Omron CX-Programmer project NewProject (CX-Programmer 9.73)

# PLC NewPLC1: CP1E N30

## Program NewProgram1 (cyclic task 0)

### Section Section1

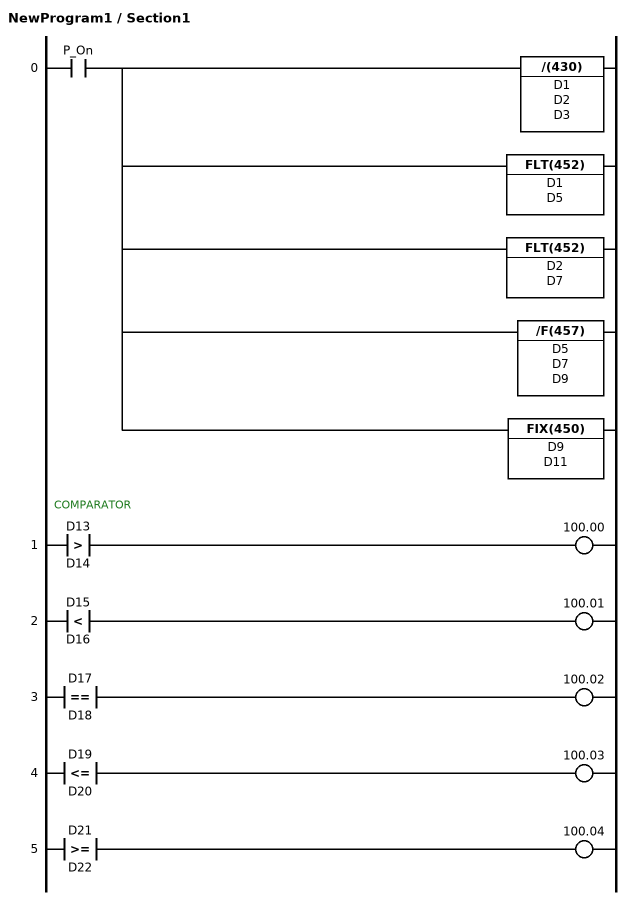
; rung 0
LD P_On
/(430) D1 D2 D3
FLT(452) D1 D5
FLT(452) D2 D7
/F(457) D5 D7 D9
FIX(450) D9 D11
; rung 1: COMPARATOR
LD>(320) D13 D14
OUT 100.00
; rung 2
LD<(310) D15 D16
OUT 100.01
; rung 3
LD=(300) D17 D18
OUT 100.02
; rung 4
LD<=(315) D19 D20
OUT 100.03
; rung 5
LD>=(325) D21 D22
OUT 100.04

### Section END
; rung 0
END(001)